Omron CX-Programmer project NewProject (CX-Programmer 9.61)

# PLC NewPLC1: CPM1(CPM1A) CPU20

## Program NewProgram1 (no task)

### Section Section1

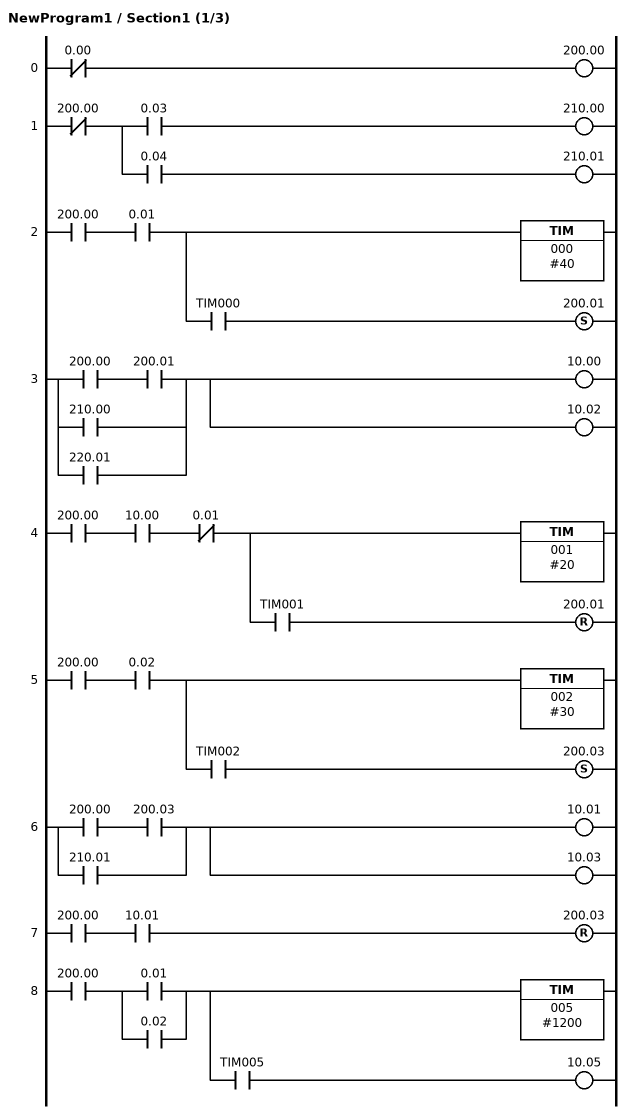
; rung 0
LDNOT 0.00
OUT 200.00
; rung 1
LDNOT 200.00
OUT TR0
AND 0.03
OUT 210.00
LD TR0
AND 0.04
OUT 210.01
; rung 2
LD 200.00
AND 0.01
TIM 000 #40
AND TIM000
SET 200.01
; rung 3
LD 200.00
AND 200.01
OR 210.00
OR 220.01
OUT 10.00
OUT 10.02
; rung 4
LD 200.00
AND 10.00
ANDNOT 0.01
TIM 001 #20
AND TIM001
RSET 200.01
; rung 5
LD 200.00
AND 0.02
TIM 002 #30
AND TIM002
SET 200.03
; rung 6
LD 200.00
AND 200.03
OR 210.01
OUT 10.01
OUT 10.03
; rung 7
LD 200.00
AND 10.01
RSET 200.03
; rung 8
LD 200.00
LD 0.01
OR 0.02
ANDLD
TIM 005 #1200
AND TIM005
OUT 10.05

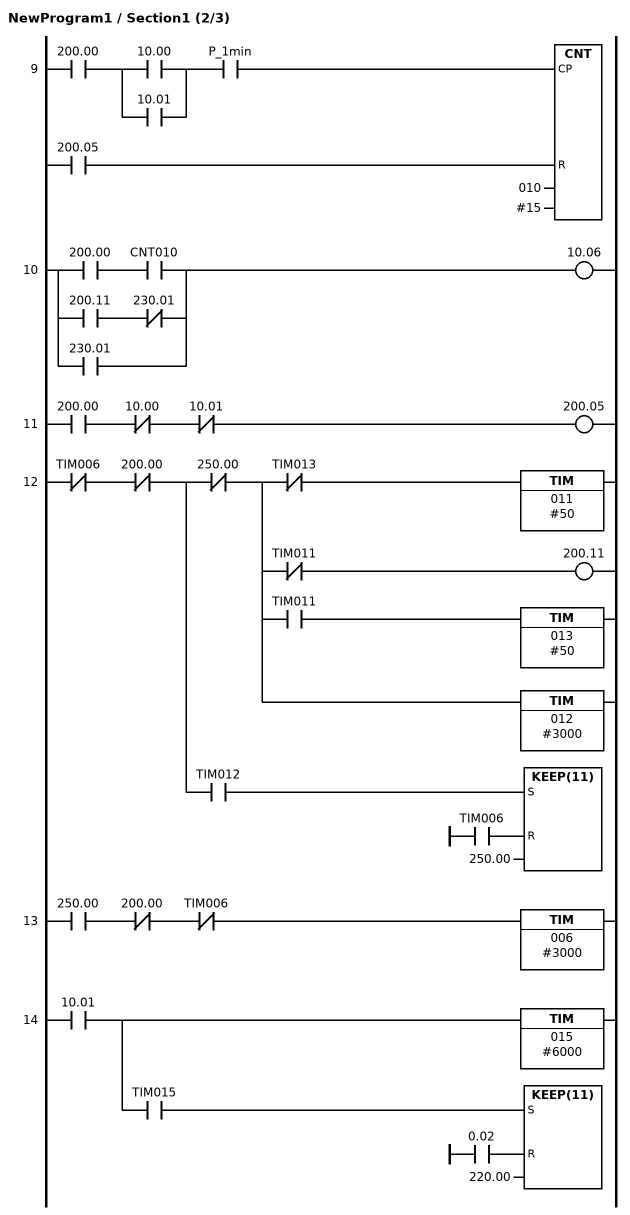
; rung 9
LD 200.00
LD 10.00
OR 10.01
ANDLD
AND P_1min
LD 200.05
CNT 010 #15
; rung 10
LD 200.00
AND CNT010
LD 200.11
ANDNOT 230.01
ORLD
OR 230.01
OUT 10.06
; rung 11
LD 200.00
ANDNOT 10.00
ANDNOT 10.01
OUT 200.05
; rung 12
LDNOT TIM006
ANDNOT 200.00
OUT TR0
ANDNOT 250.00
OUT TR1
ANDNOT TIM013
TIM 011 #50
LD TR1
ANDNOT TIM011
OUT 200.11
LD TR1
AND TIM011
TIM 013 #50
LD TR1
TIM 012 #3000
LD TR0
AND TIM012
LD TIM006
KEEP(11) 250.00
; rung 13
LD 250.00
ANDNOT 200.00
ANDNOT TIM006
TIM 006 #3000
; rung 14
LD 10.01
TIM 015 #6000
AND TIM015
LD 0.02
KEEP(11) 220.00

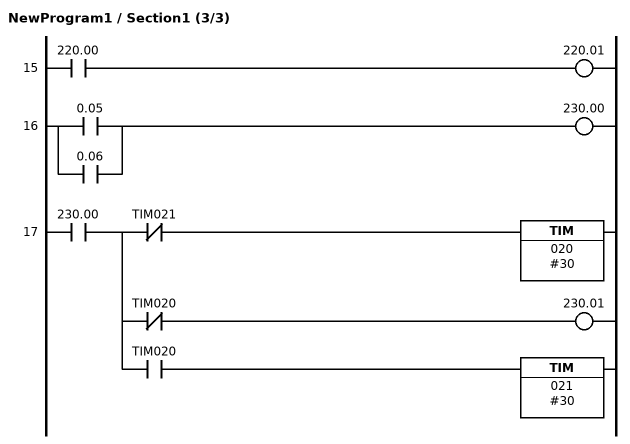
; rung 15
LD 220.00
OUT 220.01
; rung 16
LD 0.05
OR 0.06
OUT 230.00
; rung 17
LD 230.00
OUT TR0
ANDNOT TIM021
TIM 020 #30
LD TR0
ANDNOT TIM020
OUT 230.01
LD TR0
AND TIM020
TIM 021 #30

### Section Section2
; rung 0
END(01)